// TIA Portal V20 export
DATA_BLOCK "MP103"   // DB305
// stored: MemoryReserve 100
   VAR
      "ET200ECO PN-4 POWER TRIPPED E8232CB" : Bool;
      "PANEL FAN POWER TRIPPED E8304CB" : Bool;
      SPARE : Bool;
      "CONTROLLER POWER SMPS DC OK E8404PWS" : Bool;
      "CONTROLLER DC POWER TRIPPED E8406CB" : Bool;
      "KISTLER CONTROL POWER TRIPPED E8416CB" : Bool;
      "MANIFOLD-1 POWER TRIPPED E8422CB" : Bool;
      "MANIFOLD-2 POWER TRIPPED E8430CB" : Bool;
      "QR READER POWER TRIPPED E8456CB" : Bool;
      "QR READER POWER TRIPPED E8462CB" : Bool;
      "HANDY QR READER POWER TRIPPED E8468CB" : Bool;
      "PROFINET CONVERTER POWER TRIPPED E8474CB" : Bool;
      "MONITORING RELAY POWER TRIPPED E8504CB" : Bool;
      SPARE_1 : Bool;
      "SAFETY POWER SMPS DC OK E8704PWS" : Bool;
      "SAFETY DC POWER TRIPPED E8706CB" : Bool;
      "ET200SP I/O SAFETY POWER TRIPPED E8716CB" : Bool;
      "JUNCTION BOX CONTROL POWER TRIPPED E8736CB" : Bool;
      "ET200ECO PN SAFETYT-1 POWER TRIPPED E8756CB" : Bool;
      "ET200ECO PN SAFETYT-2 POWER TRIPPED E8762CB" : Bool;
      SPARE_2 : Bool;
      "CONTROL POWER SMPS DC OK E8804PWS" : Bool;
      "CONTROL DC POWER TRIPPED E8806CB" : Bool;
      "JUNCTION BOX CONTROL POWER TRIPPED E8816CB" : Bool;
      "DRIVE-CLIQ HUB POWER TRIPPED E8822CB" : Bool;
      "EQUIPMENT LED POWER TRIPPED E8828CB" : Bool;
      SPARE_3 : Bool;
      SPARE_4 : Bool;
      SPARE_5 : Bool;
      SPARE_6 : Bool;
      SPARE_7 : Bool;
      SPARE_8 : Bool;
   END_VAR
BEGIN
END_DATA_BLOCK
